TYPE ST_ScaledCylinderInputs :
STRUCT
	fPistonPressureS : LREAL;
	fRodPressureS : LREAL; 
	fCylinderPositionS : LREAL; 
END_STRUCT
END_TYPE

(* stored: Version 1.1.0.1, ProductVersion 3.1.4024.12
   DUT ST_ScaledCylinderInputs: Id {cb8712cf-fb8e-4020-b556-1e76a3c183b3} *)
